(* PLC project mtcs_hydraulics, Institute of Astronomy OntoManager 0.0.1 *)
(* stored: creationDateTime 2024-08-13T09:17:29.860254, modificationDateTime 2024-08-13T09:17:29.860254 *)

TYPE HydraulicsPumpsStates : (STOPPED := 0, POWERING_ON := 1, RESETTING_DRIVES := 2, COMMANDING_SAFETY := 3, BUILDING_UP_PRESSURE := 4, RUNNING := 5, STOPPING := 6, POWERING_OFF := 7, MANUAL := 8, ERROR := 9);
END_TYPE

TYPE HydraulicsParts : STRUCT
  circulationPumpRelay : SimpleRelay;  (* Relay to power on/off the circulation pump *)
  pumpsPowerRelay : SimpleRelay;  (* Relay to power on/off the pumps *)
  top : HydraulicsSide;  (* Top side *)
  bottom : HydraulicsSide;  (* Bottom side *)
  io : HydraulicsIO;  (* I/O modules *)
  configManager : ConfigManager;  (* The config manager (to load/save/activate configuration data) *)
END_STRUCT;
END_TYPE

TYPE HydraulicsIOParts : STRUCT
  pumpsGroup : HydraulicsPumpsGroupIO;  (* PG: Pumps Group *)
END_STRUCT;
END_TYPE

TYPE HydraulicsPumpsGroupIOParts : STRUCT
  COU : EtherCatDevice;  (* PG:COU (EK1101) *)
  DI1 : EtherCatDevice;  (* PG:DI1 (EL1008) *)
  SI1 : EtherCatDevice;  (* PG:SI1 (EL1904) *)
  SI2 : EtherCatDevice;  (* PG:SI2 (EL1904) *)
  SI3 : EtherCatDevice;  (* PG:SI3 (EL1904) *)
  DI2 : EtherCatDevice;  (* PG:DI2 (EL1008) *)
END_STRUCT;
END_TYPE

TYPE HydraulicsProcesses : STRUCT
  initialize : Process;  (* Start initializing *)
  lock : Process;  (* Lock the system *)
  unlock : Process;  (* Unlock the system *)
  changeOperatingState : ChangeOperatingStateProcess;  (* Change the operating state (e.g. AUTO, MANUAL, ...) *)
  startUpPumps : Process;  (* Start up the pumps *)
  stopPumps : Process;  (* Stop the pumps *)
END_STRUCT;
END_TYPE

TYPE HydraulicsSideProcesses : STRUCT
  resetDrive : Process;  (* Reset the drive *)
  changeFrequencySetpoint : ChangeSetpointProcess;  (* Change the frequency setpoint, in Hertz *)
END_STRUCT;
END_TYPE

TYPE HydraulicsStatuses : STRUCT
  initializationStatus : InitializationStatus;
  healthStatus : HealthStatus;
  busyStatus : BusyStatus;
  operatingStatus : OperatingStatus;
END_STRUCT;
END_TYPE

TYPE HydraulicsSideStatuses : STRUCT
  healthStatus : HealthStatus;  (* Is the hydraulics side in a healthy state? Good=RUN, Bad=safe stopped *)
  busyStatus : BusyStatus;  (* Is the hydraulics side busy? *)
END_STRUCT;
END_TYPE

TYPE HydraulicsIOStatuses : STRUCT
  healthStatus : HealthStatus;  (* Is the I/O in a healthy state? *)
END_STRUCT;
END_TYPE

TYPE HydraulicsPumpsGroupIOStatuses : STRUCT
  healthStatus : HealthStatus;  (* Is the I/O in a healthy state? *)
END_STRUCT;
END_TYPE

TYPE HydraulicsConfig : STRUCT
  top : HydraulicsSideConfig;  (* Top side settings *)
  bottom : HydraulicsSideConfig;  (* Bottom side settings *)
  controlCycleTime : LREAL;  (* Cycle time in seconds of the control loop (old system: 60.0) *)
  controlHysteresis : LREAL;  (* Don't change the frequency setpoint if the error is below this value (in Hz) (old system: 1.0) *)
  buildUpPressureTime : LREAL;  (* Time in seconds during startup, when the pumps must run at maxFrequency *)
  bearingTemperature : MeasurementConfig;  (* Oil temperature measured at the bearing *)
  stoppingTime : LREAL;  (* Time in seconds during stopping *)
  pumpsPowerOnTIme : LREAL;  (* Time in seconds to wait while powering on *)
  pumpsPowerOffTIme : LREAL;  (* Time in seconds to wait while powering off *)
END_STRUCT;
END_TYPE

TYPE HydraulicsSideConfig : STRUCT
  minFrequency : LREAL;  (* Minimum allowed frequency in Hz (old system: 50.0 for both pumps) *)
  maxFrequency : LREAL;  (* Maximum allowed frequency in Hz (old system: 100.0 for both pumps) *)
  pressureMeasurement : MeasurementConfig;  (* Pressure measurement config, in Bar *)
  pressureSensorFullScale : LREAL;  (* Sensor full scale range, in Bar *)
  frequencyMeasurement : MeasurementConfig;  (* Frequency measurement config, in Hertz *)
  frequencyMeasurementFullScale : LREAL;  (* Measurement full scale range, in Hertz *)
  conversionCoefficientA : LREAL;  (* Coefficient 'a' of formula: Frequency[Hz] = a * temp[Celsius]^2 + b * temp[Celsius] + c *)
  conversionCoefficientB : LREAL;  (* Coefficient 'b' of formula: Frequency[Hz] = a * temp[Celsius]^2 + b * temp[Celsius] + c *)
  conversionCoefficientC : LREAL;  (* Coefficient 'c' of formula: Frequency[Hz] = a * temp[Celsius]^2 + b * temp[Celsius] + c *)
END_STRUCT;
END_TYPE

FUNCTION_BLOCK SM_Hydraulics
  VAR_INPUT
    {attribute 'OPC.UA.DA' := '1'}
    {attribute 'OPC.UA.DA.Access' := '1'}
    editableConfig : HydraulicsConfig;  (* Editable configuration of the Safety subsystem *)
    {attribute 'OPC.UA.DA' := '1'}
    {attribute 'OPC.UA.DA.Access' := '1'}
    circulationFilterGOK AT %I* : BOOL;  (* TRUE if there is no overpressure for circulation filter G *)
    {attribute 'OPC.UA.DA' := '1'}
    {attribute 'OPC.UA.DA.Access' := '1'}
    circulationFilterDOK AT %I* : BOOL;  (* TRUE if there is no overpressure for circulation filter D *)
    {attribute 'OPC.UA.DA' := '1'}
    {attribute 'OPC.UA.DA.Access' := '1'}
    oilLevelTooHigh AT %I* : BOOL;  (* TRUE if the oil level is too high (--> problem!) *)
    {attribute 'OPC.UA.DA' := '1'}
    {attribute 'OPC.UA.DA.Access' := '1'}
    pumpsState : HydraulicsPumpsStates;  (* The current state of the pumps *)
    {attribute 'OPC.UA.DA' := '1'}
    {attribute 'OPC.UA.DA.Access' := '1'}
    pumpsStatus : STRING;  (* Textual representation of the current pumps status *)
  END_VAR
  VAR_OUTPUT
    {attribute 'OPC.UA.DA' := '1'}
    {attribute 'OPC.UA.DA.Access' := '1'}
    actualStatus : STRING;  (* Current status description *)
    previousStatus : STRING;  (* Previous status description *)
    {attribute 'OPC.UA.DA' := '1'}
    {attribute 'OPC.UA.DA.Access' := '1'}
    config : HydraulicsConfig;  (* Active configuration of the Hydraulics subsystem *)
    {attribute 'OPC.UA.DA' := '1'}
    {attribute 'OPC.UA.DA.Access' := '1'}
    bearingTemperature : TemperatureMeasurement;  (* Temperature measured at the bearing *)
    statuses : HydraulicsStatuses;  (* Statuses of the state machine *)
    parts : HydraulicsParts;  (* Parts of the state machine *)
    processes : HydraulicsProcesses;  (* Processes of the state machine *)
  END_VAR
  VAR_IN_OUT
    {attribute 'OPC.UA.DA' := '0'}
    operatorStatus : OperatorStatus;  (* Shared operator status *)
    {attribute 'OPC.UA.DA' := '0'}
    safetyHydraulics : SafetyHydraulics;  (* The hydraulics part of the safety system *)
    {attribute 'OPC.UA.DA' := '0'}
    safetyIO : SafetyIO;  (* The I/O part of the safety system *)
  END_VAR

            bearingTemperature( config := config.bearingTemperature );
parts.circulationPumpRelay( isEnabled := statuses.busyStatus.idle AND (operatorStatus.tech AND statuses.operatingStatus.manual) );
parts.pumpsPowerRelay( isEnabled := statuses.busyStatus.idle AND operatorStatus.tech );
parts.top(
    operatorStatus := operatorStatus,
    operatingStatus := statuses.operatingStatus,
    safetyHydraulics := safetyHydraulics,
    config := config.top,
    hydraulicsConfig := config);
parts.bottom(
    operatorStatus := operatorStatus,
    operatingStatus := statuses.operatingStatus,
    safetyHydraulics := safetyHydraulics,
    config := config.bottom,
    hydraulicsConfig := config);
parts.io( safetyIO := safetyIO );
parts.configManager( isEnabled := operatorStatus.tech );
statuses.initializationStatus();
statuses.healthStatus(
    isGood := (parts.io.statuses.healthStatus.isGood AND (parts.configManager.statuses.healthStatus.isGood AND (processes.initialize.statuses.healthStatus.isGood AND (processes.lock.statuses.healthStatus.isGood AND (processes.unlock.statuses.healthStatus.isGood AND (processes.changeOperatingState.statuses.healthStatus.isGood AND safetyHydraulics.statuses.healthStatus.isGood)))))) AND (circulationFilterGOK AND (circulationFilterDOK AND ((NOT(oilLevelTooHigh)) AND (NOT(pumpsState = HydraulicsPumpsStates.ERROR))))),
    hasWarning := (parts.io.statuses.healthStatus.hasWarning OR (parts.configManager.statuses.healthStatus.hasWarning OR (processes.initialize.statuses.healthStatus.hasWarning OR (processes.lock.statuses.healthStatus.hasWarning OR (processes.unlock.statuses.healthStatus.hasWarning OR processes.changeOperatingState.statuses.healthStatus.hasWarning))))) OR (bearingTemperature.statuses.healthStatus.hasWarning OR (bearingTemperature.statuses.healthStatus.bad OR (pumpsState = HydraulicsPumpsStates.MANUAL))));
statuses.busyStatus( isBusy := statuses.initializationStatus.initializing OR (processes.initialize.statuses.busyStatus.busy OR (processes.lock.statuses.busyStatus.busy OR (processes.unlock.statuses.busyStatus.busy OR (processes.changeOperatingState.statuses.busyStatus.busy OR (processes.startUpPumps.statuses.busyStatus.busy OR processes.stopPumps.statuses.busyStatus.busy))))) );
statuses.operatingStatus();
processes.initialize( isEnabled := statuses.initializationStatus.shutdown OR (statuses.initializationStatus.initializingFailed OR statuses.initializationStatus.initialized) );
processes.lock( isEnabled := operatorStatus.tech AND statuses.initializationStatus.initialized );
processes.unlock( isEnabled := operatorStatus.tech AND statuses.initializationStatus.locked );
processes.changeOperatingState( isEnabled := statuses.busyStatus.idle AND operatorStatus.tech );
processes.startUpPumps( isEnabled := statuses.initializationStatus.initialized AND ((pumpsState = HydraulicsPumpsStates.STOPPED) OR ((pumpsState = HydraulicsPumpsStates.MANUAL) OR (pumpsState = HydraulicsPumpsStates.ERROR))) );
processes.stopPumps( isEnabled := statuses.initializationStatus.initialized AND ((pumpsState = HydraulicsPumpsStates.RUNNING) OR ((pumpsState = HydraulicsPumpsStates.MANUAL) OR (pumpsState = HydraulicsPumpsStates.ERROR))) );

          

{attribute 'TcRpcEnable' := '1'}
METHOD initialize : RequestResults
                  initialize := THIS^.processes.initialize.request();

                
END_METHOD

{attribute 'TcRpcEnable' := '1'}
METHOD lock : RequestResults
                  lock := THIS^.processes.lock.request();

                
END_METHOD

{attribute 'TcRpcEnable' := '1'}
METHOD unlock : RequestResults
                  unlock := THIS^.processes.unlock.request();

                
END_METHOD

{attribute 'TcRpcEnable' := '1'}
METHOD changeOperatingState : RequestResults
  VAR_INPUT
    state : OperatingStates;
  END_VAR
                  changeOperatingState := THIS^.processes.changeOperatingState.request( state := state );

                
END_METHOD

{attribute 'TcRpcEnable' := '1'}
METHOD startUpPumps : RequestResults
                  startUpPumps := THIS^.processes.startUpPumps.request();

                
END_METHOD

{attribute 'TcRpcEnable' := '1'}
METHOD stopPumps : RequestResults
                  stopPumps := THIS^.processes.stopPumps.request();

                
END_METHOD

{attribute 'TcRpcEnable' := '1'}
METHOD _log : BOOL
  VAR_INPUT
    name : STRING;  (* Name of this function block instance *)
  END_VAR
  VAR_IN_OUT
    buffer : LogBuffer;  (* Buffer to write all logging to *)
  END_VAR
  VAR
    subBuffer : LogBuffer;  (* Temporary buffer to write logging by parts (sub-statemachines) to *)
  END_VAR
                  THIS^.parts.circulationPumpRelay._log(
    name := 'circulationPumpRelay',
    buffer := subBuffer);
THIS^.parts.pumpsPowerRelay._log(
    name := 'pumpsPowerRelay',
    buffer := subBuffer);
THIS^.parts.top._log(
    name := 'top',
    buffer := subBuffer);
THIS^.parts.bottom._log(
    name := 'bottom',
    buffer := subBuffer);
THIS^.parts.io._log(
    name := 'io',
    buffer := subBuffer);
THIS^.parts.configManager._log(
    name := 'configManager',
    buffer := subBuffer);
THIS^.processes.initialize._log(
    name := 'processes.initialize',
    buffer := subBuffer);
THIS^.processes.lock._log(
    name := 'processes.lock',
    buffer := subBuffer);
THIS^.processes.unlock._log(
    name := 'processes.unlock',
    buffer := subBuffer);
THIS^.processes.changeOperatingState._log(
    name := 'processes.changeOperatingState',
    buffer := subBuffer);
THIS^.processes.startUpPumps._log(
    name := 'processes.startUpPumps',
    buffer := subBuffer);
THIS^.processes.stopPumps._log(
    name := 'processes.stopPumps',
    buffer := subBuffer);
LOGGER(
    name := name,
    actualStatus := THIS^.actualStatus,
    previousStatus := THIS^.previousStatus,
    buffer := buffer,
    subBuffer := subBuffer,
    pHealthStatus := ADR(THIS^.statuses.healthStatus),
    pBusyStatus := ADR(THIS^.statuses.busyStatus));

                
END_METHOD
END_FUNCTION_BLOCK

FUNCTION_BLOCK SM_HydraulicsSide
  VAR_INPUT
    {attribute 'OPC.UA.DA' := '1'}
    {attribute 'OPC.UA.DA.Access' := '1'}
    entranceFilter1OK AT %I* : BOOL;  (* TRUE if there is no overpressure for entrance filter 1 *)
    {attribute 'OPC.UA.DA' := '1'}
    {attribute 'OPC.UA.DA.Access' := '1'}
    entranceFilter2OK AT %I* : BOOL;  (* TRUE if there is no overpressure for entrance filter 2 *)
    {attribute 'OPC.UA.DA' := '1'}
    {attribute 'OPC.UA.DA.Access' := '1'}
    entranceFilter3OK AT %I* : BOOL;  (* TRUE if there is no overpressure for entrance filter 3 *)
    {attribute 'OPC.UA.DA' := '1'}
    {attribute 'OPC.UA.DA.Access' := '1'}
    entranceFilter4OK AT %I* : BOOL;  (* TRUE if there is no overpressure for entrance filter 4 *)
  END_VAR
  VAR_OUTPUT
    {attribute 'OPC.UA.DA' := '1'}
    {attribute 'OPC.UA.DA.Access' := '1'}
    actualStatus : STRING;  (* Current status description *)
    previousStatus : STRING;  (* Previous status description *)
    {attribute 'OPC.UA.DA' := '1'}
    {attribute 'OPC.UA.DA.Access' := '1'}
    driveTripOK : BOOL;  (* TRIP output of the drive, as copied from the safety system *)
    {attribute 'OPC.UA.DA' := '1'}
    {attribute 'OPC.UA.DA.Access' := '1'}
    driveRelease : BOOL;  (* Release output of the drive (ReglerFreigabe RFR), as copied from the safety system *)
    {attribute 'OPC.UA.DA' := '1'}
    {attribute 'OPC.UA.DA.Access' := '1'}
    driveMinFrequency : BOOL;  (* Minimum frequency output of the drive (QMIN), as copied from the safety system *)
    {attribute 'OPC.UA.DA' := '1'}
    {attribute 'OPC.UA.DA.Access' := '1'}
    pressureMeasurement : PressureMeasurement;  (* Pressure measurement *)
    {attribute 'OPC.UA.DA' := '1'}
    {attribute 'OPC.UA.DA.Access' := '1'}
    frequencyMeasurement : FrequencyMeasurement;  (* Frequency measurement *)
    {attribute 'OPC.UA.DA' := '1'}
    {attribute 'OPC.UA.DA.Access' := '1'}
    driveSetpoint : Frequency;  (* Frequency setpoint actually used *)
    {attribute 'OPC.UA.DA' := '1'}
    {attribute 'OPC.UA.DA.Access' := '1'}
    driveSetpointSignal AT %Q* : INT;  (* Raw signal value of the frequency setpoint *)
    {attribute 'OPC.UA.DA' := '1'}
    {attribute 'OPC.UA.DA.Access' := '1'}
    resetDriveSignal AT %Q* : BOOL;  (* Output to reset the drive *)
    statuses : HydraulicsSideStatuses;  (* Statuses of the state machine *)
    processes : HydraulicsSideProcesses;  (* Processes of the state machine *)
  END_VAR
  VAR_IN_OUT
    {attribute 'OPC.UA.DA' := '0'}
    operatorStatus : OperatorStatus;
    {attribute 'OPC.UA.DA' := '0'}
    operatingStatus : OperatingStatus;
    {attribute 'OPC.UA.DA' := '0'}
    safetyHydraulics : SafetyHydraulics;
    {attribute 'OPC.UA.DA' := '0'}
    config : HydraulicsSideConfig;
    {attribute 'OPC.UA.DA' := '0'}
    hydraulicsConfig : HydraulicsConfig;
  END_VAR

            pressureMeasurement(
    config := config.pressureMeasurement,
    conversionFactor := config.pressureSensorFullScale / 32768.0);
frequencyMeasurement(
    config := config.frequencyMeasurement,
    conversionFactor := config.frequencyMeasurementFullScale / 32768.0);
statuses.healthStatus(
    isGood := (processes.resetDrive.statuses.healthStatus.isGood AND processes.changeFrequencySetpoint.statuses.healthStatus.isGood) AND ((pressureMeasurement.statuses.healthStatus.isGood OR pressureMeasurement.statuses.enabledStatus.disabled) AND ((frequencyMeasurement.statuses.healthStatus.isGood OR frequencyMeasurement.statuses.enabledStatus.disabled) AND (entranceFilter1OK AND (entranceFilter2OK AND (entranceFilter3OK AND (entranceFilter4OK AND driveTripOK)))))),
    hasWarning := processes.changeFrequencySetpoint.statuses.healthStatus.hasWarning OR (pressureMeasurement.statuses.healthStatus.hasWarning OR frequencyMeasurement.statuses.healthStatus.hasWarning));
statuses.busyStatus( isBusy := processes.changeFrequencySetpoint.statuses.busyStatus.busy OR processes.resetDrive.statuses.busyStatus.busy );
processes.resetDrive( isEnabled := statuses.busyStatus.idle AND operatorStatus.tech );
processes.changeFrequencySetpoint( isEnabled := statuses.busyStatus.idle AND (operatingStatus.manual AND operatorStatus.tech) );

          

{attribute 'TcRpcEnable' := '1'}
METHOD resetDrive : RequestResults
                  resetDrive := THIS^.processes.resetDrive.request();

                
END_METHOD

{attribute 'TcRpcEnable' := '1'}
METHOD changeFrequencySetpoint : RequestResults
  VAR_INPUT
    setpoint : LREAL;
  END_VAR
                  changeFrequencySetpoint := THIS^.processes.changeFrequencySetpoint.request( setpoint := setpoint );

                
END_METHOD

{attribute 'TcRpcEnable' := '1'}
METHOD _log : BOOL
  VAR_INPUT
    name : STRING;  (* Name of this function block instance *)
  END_VAR
  VAR_IN_OUT
    buffer : LogBuffer;  (* Buffer to write all logging to *)
  END_VAR
  VAR
    subBuffer : LogBuffer;  (* Temporary buffer to write logging by parts (sub-statemachines) to *)
  END_VAR
                  THIS^.processes.resetDrive._log(
    name := 'processes.resetDrive',
    buffer := subBuffer);
THIS^.processes.changeFrequencySetpoint._log(
    name := 'processes.changeFrequencySetpoint',
    buffer := subBuffer);
LOGGER(
    name := name,
    actualStatus := THIS^.actualStatus,
    previousStatus := THIS^.previousStatus,
    buffer := buffer,
    subBuffer := subBuffer,
    pHealthStatus := ADR(THIS^.statuses.healthStatus),
    pBusyStatus := ADR(THIS^.statuses.busyStatus));

                
END_METHOD
END_FUNCTION_BLOCK

FUNCTION_BLOCK SM_HydraulicsIO
  VAR_OUTPUT
    {attribute 'OPC.UA.DA' := '1'}
    {attribute 'OPC.UA.DA.Access' := '1'}
    actualStatus : STRING;  (* Current status description *)
    previousStatus : STRING;  (* Previous status description *)
    statuses : HydraulicsIOStatuses;  (* Statuses of the state machine *)
    parts : HydraulicsIOParts;  (* Parts of the state machine *)
  END_VAR
  VAR_IN_OUT
    {attribute 'OPC.UA.DA' := '0'}
    safetyIO : SafetyIO;  (* The safety I/O *)
  END_VAR

            parts.pumpsGroup();
statuses.healthStatus(
    isGood := safetyIO.statuses.healthStatus.isGood AND parts.pumpsGroup.statuses.healthStatus.isGood,
    hasWarning := safetyIO.statuses.healthStatus.hasWarning OR parts.pumpsGroup.statuses.healthStatus.hasWarning);

          

{attribute 'TcRpcEnable' := '1'}
METHOD _log : BOOL
  VAR_INPUT
    name : STRING;  (* Name of this function block instance *)
  END_VAR
  VAR_IN_OUT
    buffer : LogBuffer;  (* Buffer to write all logging to *)
  END_VAR
  VAR
    subBuffer : LogBuffer;  (* Temporary buffer to write logging by parts (sub-statemachines) to *)
  END_VAR
                  THIS^.parts.pumpsGroup._log(
    name := 'pumpsGroup',
    buffer := subBuffer);
LOGGER(
    name := name,
    actualStatus := THIS^.actualStatus,
    previousStatus := THIS^.previousStatus,
    buffer := buffer,
    subBuffer := subBuffer,
    pHealthStatus := ADR(THIS^.statuses.healthStatus));

                
END_METHOD
END_FUNCTION_BLOCK

FUNCTION_BLOCK SM_HydraulicsPumpsGroupIO
  VAR_OUTPUT
    {attribute 'OPC.UA.DA' := '1'}
    {attribute 'OPC.UA.DA.Access' := '1'}
    actualStatus : STRING;  (* Current status description *)
    previousStatus : STRING;  (* Previous status description *)
    statuses : HydraulicsPumpsGroupIOStatuses;  (* Statuses of the state machine *)
    parts : HydraulicsPumpsGroupIOParts;  (* Parts of the state machine *)
  END_VAR

            parts.COU(
    id := 'PG:COU',
    typeId := 'EK1101');
parts.DI1(
    id := 'PG:DI1',
    typeId := 'EL1008');
parts.SI1(
    id := 'PG:SI1',
    typeId := 'EL1904');
parts.SI2(
    id := 'PG:SI2',
    typeId := 'EL1904');
parts.SI3(
    id := 'PG:SI3',
    typeId := 'EL1904');
parts.DI2(
    id := 'PG:DI2',
    typeId := 'EL1008');
statuses.healthStatus(
    isGood := parts.COU.statuses.healthStatus.isGood AND (parts.DI1.statuses.healthStatus.isGood AND (parts.SI1.statuses.healthStatus.isGood AND (parts.SI2.statuses.healthStatus.isGood AND (parts.SI3.statuses.healthStatus.isGood AND parts.DI2.statuses.healthStatus.isGood)))),
    hasWarning := parts.COU.statuses.healthStatus.hasWarning OR (parts.DI1.statuses.healthStatus.hasWarning OR (parts.SI1.statuses.healthStatus.hasWarning OR (parts.SI2.statuses.healthStatus.hasWarning OR (parts.SI3.statuses.healthStatus.hasWarning OR parts.DI2.statuses.healthStatus.hasWarning)))));

          

{attribute 'TcRpcEnable' := '1'}
METHOD _log : BOOL
  VAR_INPUT
    name : STRING;  (* Name of this function block instance *)
  END_VAR
  VAR_IN_OUT
    buffer : LogBuffer;  (* Buffer to write all logging to *)
  END_VAR
  VAR
    subBuffer : LogBuffer;  (* Temporary buffer to write logging by parts (sub-statemachines) to *)
  END_VAR
                  THIS^.parts.COU._log(
    name := 'COU',
    buffer := subBuffer);
THIS^.parts.DI1._log(
    name := 'DI1',
    buffer := subBuffer);
THIS^.parts.SI1._log(
    name := 'SI1',
    buffer := subBuffer);
THIS^.parts.SI2._log(
    name := 'SI2',
    buffer := subBuffer);
THIS^.parts.SI3._log(
    name := 'SI3',
    buffer := subBuffer);
THIS^.parts.DI2._log(
    name := 'DI2',
    buffer := subBuffer);
LOGGER(
    name := name,
    actualStatus := THIS^.actualStatus,
    previousStatus := THIS^.previousStatus,
    buffer := buffer,
    subBuffer := subBuffer,
    pHealthStatus := ADR(THIS^.statuses.healthStatus));

                
END_METHOD
END_FUNCTION_BLOCK
